PROGRAM MAIN
VAR

END_VAR

END_PROGRAM

(* stored: Version 1.1.0.1, ProductVersion 3.1.4024.12
   POU MAIN: Id {cb0dada2-790f-48b3-8702-fc17bd7e66f5}, SpecialFunc None *)
